ABB RAPID module: Module1.modx

MODULE Module1
    !***********************************************************
    !
    ! Module:  Module1
    !
    ! Description:
    !   <Insert description here>
    !
    ! Author: sm7174
    !
    ! Version: 1.0
    !
    !***********************************************************


    !***********************************************************
    !
    ! Procedure main
    !
    !   This is the entry point of your program
    !
    !***********************************************************
    PROC main()
        Ex001_Run;
        Ex002_Run;
        Ex003_Run;
        Ex004_Run;
        Ex005_Run;
    ENDPROC
ENDMODULE
